{attribute 'qualified_only'}
VAR_GLOBAL
    manager      : Forceables;
    arrForceables : ARRAY[0..MAXFORCEABLES - 1] OF ST_ForceAble;
END_VAR

VAR_GLOBAL CONSTANT
    MAXFORCEABLES : INT := 100;
END_VAR

(* stored: Version 1.1.0.1, ProductVersion 3.1.4026.18
   GVL GVL_Forceables: Id {96a6344b-f85c-4be6-b413-6e363ba9f5e3} *)
